Universal Robots PolyScope program: Colaborativo_Equipo8.urp

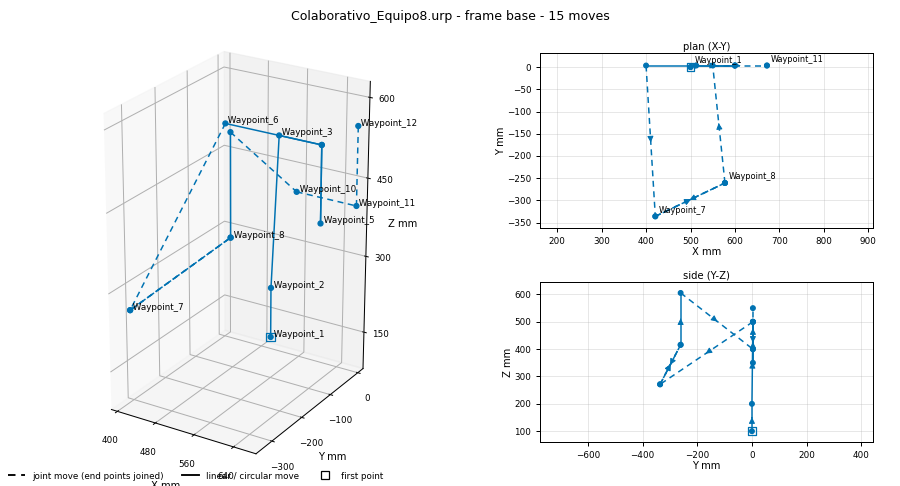
[picture p0: tool path of Colaborativo_Equipo8.urp in frame base, 15 of 15 moves have a stored position in this frame; points joined in program order, loops and branches not executed]
Program Colaborativo_Equipo8 (installation=default directory=/home/hugo/Documents/Proyecto_Ingenieria/ursim-5.10.2.106319/programs/ASM/Clase4_ActividadPractica createdIn=5.10.2.106319 lastSavedIn=5.10.2.106319 robotSerialNumber=20195599999)
Calibrated DH parameters: a=[0, -0.425, -0.3922, 0, 0, 0]; d=[0.1625, 0, 0, 0.1333, 0.0997, 0.0996]; alpha=[1.570796, 0, 0, 1.570796, -1.570796, 0]; deltaTheta=[0, 0, 0, 0, 0, 0]
Robot Program (runOnlyOnce=false)
  MoveL speed 250 mm/s, acceleration 1200 mm/s^2 (useActiveTCP=true) feature=Base
    Waypoint Waypoint_1: TCP in base x=500 y=0 z=100 mm, rx=0 ry=3.14 rz=0 rad; joints [15.467, -116.733, -124.147, -29.032, 89.976, 105.467] deg
    Waypoint Waypoint_2: TCP in base x=500 y=0 z=200 mm, rx=0 ry=3.14 rz=0 rad; joints [15.467, -104.001, -120.608, -45.303, 89.976, 105.467] deg
    Waypoint Waypoint_3: TCP in base x=512.833 y=3.551 z=500 mm, rx=0 ry=3.14 rz=0 rad; joints [15.467, -90.45, -87.803, -91.66, 89.976, 105.467] deg
    Waypoint Waypoint_4: TCP in base x=600 y=3.551 z=500 mm, rx=0 ry=3.14 rz=0 rad; joints [13.179, -102.722, -74.007, -93.182, 89.979, 103.179] deg
    Waypoint Waypoint_5: TCP in base x=600 y=3.551 z=350 mm, rx=0 ry=3.14 rz=0 rad; joints [13.179, -105.376, -92.877, -71.658, 89.979, 103.179] deg
    Waypoint Waypoint_4: TCP in base x=600 y=3.551 z=500 mm, rx=0 ry=3.14 rz=0 rad; joints [13.179, -102.722, -74.007, -93.182, 89.979, 103.179] deg
    Waypoint Waypoint_6: TCP in base x=400 y=3.551 z=500 mm, rx=0 ry=3.14 rz=0 rad; joints [19.982, -74.448, -101.53, -93.937, 89.969, 109.982] deg
  MoveJ speed 60 deg/s, acceleration 80 deg/s^2 (useActiveTCP=true) feature=Base
    Waypoint Waypoint_7: TCP in base x=420.8 y=-335.799 z=271.417 mm, rx=0.1389 ry=-2.2029 rz=2.1144 rad; joints [-13.285, -124.67, -113.908, 48.496, 13.577, 2.679] deg
    Waypoint Waypoint_8: TCP in base x=577.485 y=-260.679 z=415.906 mm, rx=0.6707 ry=1.708 rz=-1.5783 rad; joints [-2.923, -122.918, -88.146, 29.216, 11.53, 53.289] deg
  MoveJ speed 60 deg/s, acceleration 80 deg/s^2 (useActiveTCP=true) feature=Base
    Waypoint Waypoint_7: TCP in base x=420.8 y=-335.799 z=271.417 mm, rx=0.1389 ry=-2.2029 rz=2.1144 rad; joints [-13.285, -124.67, -113.908, 48.496, 13.577, 2.679] deg
    Waypoint Waypoint_8: TCP in base x=577.485 y=-260.679 z=415.906 mm, rx=0.6707 ry=1.708 rz=-1.5783 rad; joints [-2.923, -122.918, -88.146, 29.216, 11.53, 53.289] deg
  MoveL speed 250 mm/s, acceleration 1200 mm/s^2 (useActiveTCP=true) feature=Base
    Waypoint Waypoint_9: TCP in base x=577.485 y=-260.679 z=605.49 mm, rx=0.6707 ry=1.708 rz=-1.5783 rad; joints [-2.923, -114.614, -71.592, 4.359, 11.53, 53.289] deg
  MoveJ speed 60 deg/s, acceleration 80 deg/s^2 (useActiveTCP=true) feature=Base
    Waypoint Waypoint_10: TCP in base x=550 y=3.551 z=400 mm, rx=0 ry=3.14 rz=0 rad; joints [14.4, -96.875, -95.642, -77.395, 89.977, 104.4] deg
    Waypoint Waypoint_11: TCP in base x=671.952 y=3.551 z=400 mm, rx=0 ry=3.14 rz=0 rad; joints [11.748, -113.59, -74.109, -82.212, 89.981, 101.747] deg
    Waypoint Waypoint_12: TCP in base x=671.952 y=3.551 z=550 mm, rx=0 ry=3.14 rz=0 rad; joints [11.748, -115.062, -49.87, -104.979, 89.981, 101.747] deg
    Halt
